(* IEC 61131-3 sources: repolevel_ST_code_completion/output/full_case_fixed/repoeval_barrier/readful_result_history, 48 files *)

(* ---- CAN_Read_Data_SWMC_0.st ---- *)
FUNCTION CAN_Read_Data_SWMC : Can_baseframe
VAR_INPUT
	SWMC_ID	 :UINT;		//接收SWMC控制ID
	I	 	 :UINT;      //接收缓冲区域
END_VAR
VAR
	frame : Can_baseframe;
END_VAR

CASE SWMC_ID OF
	1: // SWMC-C1
		frame.id := (gCan.C1RxMsg.RXMsg[I].RxMsg_CobId - 8) / 32;
		frame.data := gCan.C1RxMsg.RXMsg[I].RxMsg_Byte;
	2: // SWMC-C2
		frame.id := (gCan.C2RxMsg.RXMsg[I].RxMsg_CobId - 8) / 32;
		frame.data := gCan.C2RxMsg.RXMsg[I].RxMsg_Byte;
	3: // SWMC-C3
		frame.id := (gCan.C3RxMsg.RXMsg[I].RxMsg_CobId - 8) / 32;
		frame.data := gCan.C3RxMsg.RXMsg[I].RxMsg_Byte;
	4: // SWMC-C4
		frame.id := (gCan.C4RxMsg.RXMsg[I].RxMsg_CobId - 8) / 32;
		frame.data := gCan.C4RxMsg.RXMsg[I].RxMsg_Byte;
	5: // SWMC-C5
		frame.id := (gCan.C5RxMsg.RXMsg[I].RxMsg_CobId - 8) / 32;
		frame.data := gCan.C5RxMsg.RXMsg[I].RxMsg_Byte;
	6: // SWMC-C6
		frame.id := (gCan.C6RxMsg.RXMsg[I].RxMsg_CobId - 8) / 32;
		frame.data := gCan.C6RxMsg.RXMsg[I].RxMsg_Byte;
	ELSE // Other
		frame.id := 0;
		frame.data[1] := 0;
		frame.data[2] := 0;
		frame.data[3] := 0;
		frame.data[4] := 0;
		frame.data[5] := 0;
		frame.data[6] := 0;
		frame.data[7] := 0;
END_CASE;

RETURN frame;
END_FUNCTION

(* ---- CAN_Read_Data_SWMC_1.st ---- *)
FUNCTION CAN_Read_Data_SWMC : Can_baseframe
VAR_INPUT
  SWMC_ID	 :UINT;		//接收SWMC控制ID
  I	 	 :UINT;      //接收缓冲区域
END_VAR
VAR
  frame : Can_baseframe;
END_VAR

CASE SWMC_ID OF
  1: // SWMC-C1
    frame.id := (gCan.C1RxMsg.RXMsg[I].RxMsg_CobId - 8) / 32;
    frame.data := gCan.C1RxMsg.RXMsg[I].RxMsg_Byte;
  2: // SWMC-C2
    frame.id := (gCan.C2RxMsg.RXMsg[I].RxMsg_CobId - 8) / 32;
    frame.data := gCan.C2RxMsg.RXMsg[I].RxMsg_Byte;
  3: // SWMC-C3
    frame.id := (gCan.C3RxMsg.RXMsg[I].RxMsg_CobId - 8) / 32;
    frame.data := gCan.C3RxMsg.RXMsg[I].RxMsg_Byte;
  4: // SWMC-C4
    frame.id := (gCan.C4RxMsg.RXMsg[I].RxMsg_CobId - 8) / 32;
    frame.data := gCan.C4RxMsg.RXMsg[I].RxMsg_Byte;
  5: // SWMC-C5
    frame.id := (gCan.C5RxMsg.RXMsg[I].RxMsg_CobId - 8) / 32;
    frame.data := gCan.C5RxMsg.RXMsg[I].RxMsg_Byte;
  6: // SWMC-C6
    frame.id := (gCan.C6RxMsg.RXMsg[I].RxMsg_CobId - 8) / 32;
    frame.data := gCan.C6RxMsg.RXMsg[I].RxMsg_Byte;
  ELSE // Other
    frame.id := 0;
    frame.data := [0, 0, 0, 0, 0, 0, 0, 0];
END_CASE;

// Explicitly return the frame structure in ST functions
CAN_Read_Data_SWMC := frame;
END_FUNCTION

(* ---- CAN_Read_Data_SWMC_2.st ---- *)
FUNCTION CAN_Read_Data_SWMC : Can_baseframe
VAR_INPUT
 SWMC_ID	 :UINT;		//接收SWMC控制ID
 I	 	 :UINT;      //接收缓冲区域
END_VAR
VAR
 frame : Can_baseframe;
END_VAR

CASE SWMC_ID OF
 1: // SWMC-C1
  frame.id := (gCan.C1RxMsg.RXMsg[I].RxMsg_CobId - 8) / 32;
  frame.data := gCan.C1RxMsg.RXMsg[I].RxMsg_Byte;
 2: // SWMC-C2
  frame.id := (gCan.C2RxMsg.RXMsg[I].RxMsg_CobId - 8) / 32;
  frame.data := gCan.C2RxMsg.RXMsg[I].RxMsg_Byte;
 3: // SWMC-C3
  frame.id := (gCan.C3RxMsg.RXMsg[I].RxMsg_CobId - 8) / 32;
  frame.data := gCan.C3RxMsg.RXMsg[I].RxMsg_Byte;
 4: // SWMC-C4
  frame.id := (gCan.C4RxMsg.RXMsg[I].RxMsg_CobId - 8) / 32;
  frame.data := gCan.C4RxMsg.RXMsg[I].RxMsg_Byte;
 5: // SWMC-C5
  frame.id := (gCan.C5RxMsg.RXMsg[I].RxMsg_CobId - 8) / 32;
  frame.data := gCan.C5RxMsg.RXMsg[I].RxMsg_Byte;
 6: // SWMC-C6
  frame.id := (gCan.C6RxMsg.RXMsg[I].RxMsg_CobId - 8) / 32;
  frame.data := gCan.C6RxMsg.RXMsg[I].RxMsg_Byte;
 ELSE // Other
  frame.id := 0;
  frame.data[0] := 0; // Element-wise assignment
  frame.data[1] := 0;
  frame.data[2] := 0;
  frame.data[3] := 0;
  frame.data[4] := 0;
  frame.data[5] := 0;
  frame.data[6] := 0;
  frame.data[7] := 0;
END_CASE;

// Explicitly return the frame structure in ST functions
CAN_Read_Data_SWMC := frame;
END_FUNCTION

(* ---- CAN_Send_Data_SWMC_0.st ---- *)
FUNCTION CAN_Send_Data_SWMC : BOOL
VAR_INPUT
	SWMC_ID : UINT;
	id 		: UINT;
	data	: ARRAY[1..8] OF BYTE;
END_VAR
VAR
	result : BOOL := FALSE;
END_VAR

CASE SWMC_ID OF
	1:
		gCan.C1TxMsg.TXMsg[1].TxMsg_CobId := 8 + 32 * id;
		gCan.C1TxMsg.TXMsg[1].TxMsg_Byte := data;
		gCan.C1TxMsg.NoOfTxMessages := 1;
		gCan.C1TxMsg.TxCounter := gCan.C1TxMsg.TxCounter + 1;
		result := TRUE;
	2:
		gCan.C2TxMsg.TXMsg[1].TxMsg_CobId := 8 + 32 * id;
		gCan.C2TxMsg.TXMsg[1].TxMsg_Byte := data;
		gCan.C2TxMsg.NoOfTxMessages := 1;
		gCan.C2TxMsg.TxCounter := gCan.C2TxMsg.TxCounter + 1;
		result := TRUE;
	3:
		gCan.C3TxMsg.TXMsg[1].TxMsg_CobId := 8 + 32 * id;
		gCan.C3TxMsg.TXMsg[1].TxMsg_Byte := data;
		gCan.C3TxMsg.NoOfTxMessages := 1;
		gCan.C3TxMsg.TxCounter := gCan.C3TxMsg.TxCounter + 1;
		result := TRUE;
	4:
		gCan.C4TxMsg.TXMsg[1].TxMsg_CobId := 8 + 32 * id;
		gCan.C4TxMsg.TXMsg[1].TxMsg_Byte := data;
		gCan.C4TxMsg.NoOfTxMessages := 1;
		gCan.C4TxMsg.TxCounter := gCan.C4TxMsg.TxCounter + 1;
		result := TRUE;
	ELSE
		result := FALSE;
END_CASE;

RETURN result;
END_FUNCTION

(* ---- CAN_Send_Data_SWMC_2.st ---- *)
FUNCTION CAN_Send_Data_SWMC : BOOL
VAR_INPUT
	SWMC_ID : UINT;
	id 		: UINT;
	data	: ARRAY[1..8] OF BYTE;
END_VAR
VAR
	result : BOOL := FALSE;
END_VAR

CASE SWMC_ID OF
	1:
		gCan.C1TxMsg.TXMsg[1].TxMsg_CobId := 8 + 32 * id;
		gCan.C1TxMsg.TXMsg[1].TxMsg_Byte := data;
		gCan.C1TxMsg.NoOfTxMessages := 1;
		gCan.C1TxMsg.TxCounter := gCan.C1TxMsg.TxCounter + 1;
		result := TRUE;
	2:
		gCan.C2TxMsg.TXMsg[1].TxMsg_CobId := 8 + 32 * id;
		gCan.C2TxMsg.TXMsg[1].TxMsg_Byte := data;
		gCan.C2TxMsg.NoOfTxMessages := 1;
		gCan.C2TxMsg.TxCounter := gCan.C2TxMsg.TxCounter + 1;
		result := TRUE;
	3:
		gCan.C3TxMsg.TXMsg[1].TxMsg_CobId := 8 + 32 * id;
		gCan.C3TxMsg.TXMsg[1].TxMsg_Byte := data;
		gCan.C3TxMsg.NoOfTxMessages := 1;
		gCan.C3TxMsg.TxCounter := gCan.C3TxMsg.TxCounter + 1;
		result := TRUE;
	4:
		gCan.C4TxMsg.TXMsg[1].TxMsg_CobId := 8 + 32 * id;
		gCan.C4TxMsg.TXMsg[1].TxMsg_Byte := data;
		gCan.C4TxMsg.NoOfTxMessages := 1;
		gCan.C4TxMsg.TxCounter := gCan.C4TxMsg.TxCounter + 1;
		result := TRUE;
	ELSE
		result := FALSE;
END_CASE;

RETURN result;
END_FUNCTION

(* ---- CAN_Send_Data_SWMC_3.st ---- *)
FUNCTION CAN_Send_Data_SWMC : BOOL
VAR_INPUT
	SWMC_ID : UINT;
	id 		: UINT;
	data	: ARRAY[1..8] OF BYTE;
END_VAR
VAR
	result : BOOL := FALSE;
END_VAR

CASE SWMC_ID OF
	1:
		gCan.C1TxMsg.TXMsg[1].TxMsg_CobId := 8 + 32 * id;
		gCan.C1TxMsg.TXMsg[1].TxMsg_Byte := data;
		gCan.C1TxMsg.NoOfTxMessages := 1;
		gCan.C1TxMsg.TxCounter := gCan.C1TxMsg.TxCounter + 1;
		result := TRUE;
	2:
		gCan.C2TxMsg.TXMsg[1].TxMsg_CobId := 8 + 32 * id;
		gCan.C2TxMsg.TXMsg[1].TxMsg_Byte := data;
		gCan.C2TxMsg.NoOfTxMessages := 1;
		gCan.C2TxMsg.TxCounter := gCan.C2TxMsg.TxCounter + 1;
		result := TRUE;
	3:
		gCan.C3TxMsg.TXMsg[1].TxMsg_CobId := 8 + 32 * id;
		gCan.C3TxMsg.TXMsg[1].TxMsg_Byte := data;
		gCan.C3TxMsg.NoOfTxMessages := 1;
		gCan.C3TxMsg.TxCounter := gCan.C3TxMsg.TxCounter + 1;
		result := TRUE;
	4:
		gCan.C4TxMsg.TXMsg[1].TxMsg_CobId := 8 + 32 * id;
		gCan.C4TxMsg.TXMsg[1].TxMsg_Byte := data;
		gCan.C4TxMsg.NoOfTxMessages := 1;
		gCan.C4TxMsg.TxCounter := gCan.C4TxMsg.TxCounter + 1;
		result := TRUE;
	ELSE
		result := FALSE;
END_CASE;

RETURN result;
END_FUNCTION

(* ---- DataReverse_cmdReverse_0.st ---- *)
FUNCTION cmdReverse : TargetDirect
VAR_INPUT
	input		:TargetDirect;
END_VAR
IF input = TargetDirect.extend THEN
	cmdReverse := TargetDirect.retract;
ELSIF input = TargetDirect.retract THEN
	cmdReverse := TargetDirect.extend;
ELSE
	cmdReverse := input; // Default case if input is neither extend nor retract
END_IF;
RETURN;
END_FUNCTION

(* ---- DataReverse_cmdReverse_1.st ---- *)
FUNCTION cmdReverse : TargetDirect
VAR_INPUT
  input		:TargetDirect;
END_VAR
IF input = TargetDirect.extend THEN
  cmdReverse := TargetDirect.retract;
ELSIF input = TargetDirect.retract THEN
  cmdReverse := TargetDirect.extend;
ELSE
  cmdReverse := input; // Default case if input is neither extend nor retract
END_IF;
END_FUNCTION

(* ---- DataReverse_cmdReverse_2.st ---- *)
FUNCTION cmdReverse : TargetDirect
VAR_INPUT
 input		:TargetDirect;
END_VAR
IF input = TargetDirect.extend THEN
 cmdReverse := TargetDirect.retract;
ELSIF input = TargetDirect.retract THEN
 cmdReverse := TargetDirect.extend;
ELSE
 cmdReverse := input; // Default case if input is neither extend nor retract
END_IF;
RETURN;
END_FUNCTION

(* ---- DataReverse_cmdReverse_3.st ---- *)
FUNCTION cmdReverse : TargetDirect
VAR_INPUT
input		:TargetDirect;
END_VAR
IF input = TargetDirect.extend THEN
cmdReverse := TargetDirect.retract;
ELSIF input = TargetDirect.retract THEN
cmdReverse := TargetDirect.extend;
ELSE
cmdReverse := input; // Default case if input is neither extend nor retract
END_IF;
RETURN;
END_FUNCTION

(* ---- setButtonByDirect_0.st ---- *)
FUNCTION setButtonByDirect : BOOL
VAR_INPUT
	level		:INT;	//1->地轨	2->天轨
	idx			:INT;	//挡板索引编号
	direct		:TargetDirect;
END_VAR
VAR
END_VAR

CASE level OF
	1:
		IF idx = 0 OR idx > 10 THEN		//参数校验
			RETURN;
		END_IF
		CASE direct OF
			TargetDirect.extend:
				gUI.grd[idx].btnStop := FALSE;
				gUI.grd[idx].btnExtend := TRUE;
				gUI.grd[idx].btnRetract := FALSE;
			TargetDirect.retract:
				gUI.grd[idx].btnStop := FALSE;
				gUI.grd[idx].btnExtend := FALSE;
				gUI.grd[idx].btnRetract := TRUE;
			TargetDirect.stop:
				gUI.grd[idx].btnStop := TRUE;
				gUI.grd[idx].btnExtend := FALSE;
				gUI.grd[idx].btnRetract := FALSE;
		END_CASE
	2:
		IF idx = 0 OR idx > 10 THEN		//参数校验
			RETURN;
		END_IF
		CASE direct OF
			TargetDirect.extend:
				gUI.sky[idx].btnStop := FALSE;
				gUI.sky[idx].btnExtend := TRUE;
				gUI.sky[idx].btnRetract := FALSE;
			TargetDirect.retract:
				gUI.sky[idx].btnStop := FALSE;
				gUI.sky[idx].btnExtend := FALSE;
				gUI.sky[idx].btnRetract := TRUE;
			TargetDirect.stop:
				gUI.sky[idx].btnStop := TRUE;
				gUI.sky[idx].btnExtend := FALSE;
				gUI.sky[idx].btnRetract := FALSE;
		END_CASE
END_CASE

RETURN;
END_FUNCTION

(* ---- setButtonByDirect_1.st ---- *)
FUNCTION setButtonByDirect : BOOL
VAR_INPUT
	level		:INT;	//1->地轨	2->天轨
	idx			:INT;	//挡板索引编号
	direct		:TargetDirect;
END_VAR
VAR
END_VAR

CASE level OF
	1:
		IF idx = 0 OR idx > 10 THEN		//参数校验
			RETURN;
		END_IF
		CASE direct OF
			TargetDirect.extend:
				gUI.grd[idx].btnStop := FALSE;
				gUI.grd[idx].btnExtend := TRUE;
				gUI.grd[idx].btnRetract := FALSE;
			TargetDirect.retract:
				gUI.grd[idx].btnStop := FALSE;
				gUI.grd[idx].btnExtend := FALSE;
				gUI.grd[idx].btnRetract := TRUE;
			TargetDirect.stop:
				gUI.grd[idx].btnStop := TRUE;
				gUI.grd[idx].btnExtend := FALSE;
				gUI.grd[idx].btnRetract := FALSE;
		END_CASE
	2:
		IF idx = 0 OR idx > 10 THEN		//参数校验
			RETURN;
		END_IF
		CASE direct OF
			TargetDirect.extend:
				gUI.sky[idx].btnStop := FALSE;
				gUI.sky[idx].btnExtend := TRUE;
				gUI.sky[idx].btnRetract := FALSE;
			TargetDirect.retract:
				gUI.sky[idx].btnStop := FALSE;
				gUI.sky[idx].btnExtend := FALSE;
				gUI.sky[idx].btnRetract := TRUE;
			TargetDirect.stop:
				gUI.sky[idx].btnStop := TRUE;
				gUI.sky[idx].btnExtend := FALSE;
				gUI.sky[idx].btnRetract := FALSE;
		END_CASE
END_CASE

RETURN;
END_FUNCTION

(* ---- setButtonByDirect_2.st ---- *)
FUNCTION setButtonByDirect : BOOL
VAR_INPUT
	level		:INT;	//1->地轨	2->天轨
	idx			:INT;	//挡板索引编号
	direct		:TargetDirect;
END_VAR
VAR
END_VAR

CASE level OF
	1:
		IF idx = 0 OR idx > 10 THEN		//参数校验
			RETURN;
		END_IF
		CASE direct OF
			TargetDirect.extend:
				gUI.grd[idx].btnStop := FALSE;
				gUI.grd[idx].btnExtend := TRUE;
				gUI.grd[idx].btnRetract := FALSE;
			TargetDirect.retract:
				gUI.grd[idx].btnStop := FALSE;
				gUI.grd[idx].btnExtend := FALSE;
				gUI.grd[idx].btnRetract := TRUE;
			TargetDirect.stop:
				gUI.grd[idx].btnStop := TRUE;
				gUI.grd[idx].btnExtend := FALSE;
				gUI.grd[idx].btnRetract := FALSE;
		END_CASE
	2:
		IF idx = 0 OR idx > 10 THEN		//参数校验
			RETURN;
		END_IF
		CASE direct OF
			TargetDirect.extend:
				gUI.sky[idx].btnStop := FALSE;
				gUI.sky[idx].btnExtend := TRUE;
				gUI.sky[idx].btnRetract := FALSE;
			TargetDirect.retract:
				gUI.sky[idx].btnStop := FALSE;
				gUI.sky[idx].btnExtend := FALSE;
				gUI.sky[idx].btnRetract := TRUE;
			TargetDirect.stop:
				gUI.sky[idx].btnStop := TRUE;
				gUI.sky[idx].btnExtend := FALSE;
				gUI.sky[idx].btnRetract := FALSE;
		END_CASE
END_CASE

RETURN;
END_FUNCTION

(* ---- setButtonByDirect_3.st ---- *)
FUNCTION setButtonByDirect : BOOL
VAR_INPUT
	level		:INT;	//1->地轨	2->天轨
	idx			:INT;	//挡板索引编号
	direct		:TargetDirect;
END_VAR
VAR
END_VAR

CASE level OF
	1:
		IF idx = 0 OR idx > 10 THEN		//参数校验
			RETURN;
		END_IF
		CASE direct OF
			TargetDirect.extend:
				gUI.grd[idx].btnStop := FALSE;
				gUI.grd[idx].btnExtend := TRUE;
				gUI.grd[idx].btnRetract := FALSE;
			TargetDirect.retract:
				gUI.grd[idx].btnStop := FALSE;
				gUI.grd[idx].btnExtend := FALSE;
				gUI.grd[idx].btnRetract := TRUE;
			TargetDirect.stop:
				gUI.grd[idx].btnStop := TRUE;
				gUI.grd[idx].btnExtend := FALSE;
				gUI.grd[idx].btnRetract := FALSE;
		END_CASE
	2:
		IF idx = 0 OR idx > 10 THEN		//参数校验
			RETURN;
		END_IF
		CASE direct OF
			TargetDirect.extend:
				gUI.sky[idx].btnStop := FALSE;
				gUI.sky[idx].btnExtend := TRUE;
				gUI.sky[idx].btnRetract := FALSE;
			TargetDirect.retract:
				gUI.sky[idx].btnStop := FALSE;
				gUI.sky[idx].btnExtend := FALSE;
				gUI.sky[idx].btnRetract := TRUE;
			TargetDirect.stop:
				gUI.sky[idx].btnStop := TRUE;
				gUI.sky[idx].btnExtend := FALSE;
				gUI.sky[idx].btnRetract := FALSE;
		END_CASE
END_CASE

RETURN;
END_FUNCTION

(* ---- CommandExecutor0_0.st ---- *)
FUNCTION_BLOCK CommandExecutor0
VAR_INPUT
	level		:INT;			//1->地轨	2->天轨
	idx			:INT;			//挡板索引编号
	direct		:TargetDirect;	//方向
	percent		:REAL;			//比例阀百分比 传入0-100
END_VAR
VAR_OUTPUT
END_VAR
VAR
END_VAR

CASE direct OF
	TargetDirect.extend:
		CASE level OF
			1:
				gController.grd[idx].extendPercent := REAL_TO_WORD(percent * 65535 / 100);
				gController.grd[idx].retractPercent := 0;
			2:
				gController.sky[idx].extendPercent := REAL_TO_WORD(percent * 65535 / 100);
				gController.sky[idx].retractPercent := 0;
		END_CASE
	TargetDirect.retract:
		CASE level OF
			1:
				gController.grd[idx].extendPercent := 0;
				gController.grd[idx].retractPercent := REAL_TO_WORD(percent * 65535 / 100);
			2:
				gController.sky[idx].extendPercent := 0;
				gController.sky[idx].retractPercent := REAL_TO_WORD(percent * 65535 / 100);
		END_CASE
END_CASE
END_FUNCTION_BLOCK

(* ---- CommandExecutor0_1.st ---- *)
FUNCTION_BLOCK CommandExecutor0
VAR_INPUT
	level		:INT;			//1->地轨	2->天轨
	idx			:INT;			//挡板索引编号
	direct		:TargetDirect;	//方向
	percent		:REAL;			//比例阀百分比 传入0-100
END_VAR
VAR_OUTPUT
END_VAR
VAR
END_VAR

CASE direct OF
	TargetDirect.extend:
		CASE level OF
			1:
				gController.grd[idx].extendPercent := REAL_TO_WORD(percent * 65535 / 100);
				gController.grd[idx].retractPercent := 0;
			2:
				gController.sky[idx].extendPercent := REAL_TO_WORD(percent * 65535 / 100);
				gController.sky[idx].retractPercent := 0;
		END_CASE
	TargetDirect.retract:
		CASE level OF
			1:
				gController.grd[idx].extendPercent := 0;
				gController.grd[idx].retractPercent := REAL_TO_WORD(percent * 65535 / 100);
			2:
				gController.sky[idx].extendPercent := 0;
				gController.sky[idx].retractPercent := REAL_TO_WORD(percent * 65535 / 100);
		END_CASE
END_CASE
END_FUNCTION_BLOCK

(* ---- CommandExecutor0_2.st ---- *)
FUNCTION_BLOCK CommandExecutor0
VAR_INPUT
	level		:INT;			//1->地轨	2->天轨
	idx			:INT;			//挡板索引编号
	direct		:TargetDirect;	//方向
	percent		:REAL;			//比例阀百分比 传入0-100
END_VAR
VAR_OUTPUT
END_VAR
VAR
END_VAR

CASE direct OF
  TargetDirect.extend:
    CASE level OF
      1:
        IF (idx >= 0) AND (idx < SIZEOF(gController.grd)) THEN
          IF (percent >= 0) AND (percent <= 100) THEN
            gController.grd[idx].extendPercent := REAL_TO_WORD(percent * 65535 / 100);
            gController.grd[idx].retractPercent := 0;
          END_IF;
        END_IF;
      2:
        IF (idx >= 0) AND (idx < SIZEOF(gController.sky)) THEN
          IF (percent >= 0) AND (percent <= 100) THEN
            gController.sky[idx].extendPercent := REAL_TO_WORD(percent * 65535 / 100);
            gController.sky[idx].retractPercent := 0;
          END_IF;
        END_IF;
    END_CASE
  TargetDirect.retract:
    CASE level OF
      1:
        IF (idx >= 0) AND (idx < SIZEOF(gController.grd)) THEN
          IF (percent >= 0) AND (percent <= 100) THEN
            gController.grd[idx].extendPercent := 0;
            gController.grd[idx].retractPercent := REAL_TO_WORD(percent * 65535 / 100);
          END_IF;
        END_IF;
      2:
        IF (idx >= 0) AND (idx < SIZEOF(gController.sky)) THEN
          IF (percent >= 0) AND (percent <= 100) THEN
            gController.sky[idx].extendPercent := 0;
            gController.sky[idx].retractPercent := REAL_TO_WORD(percent * 65535 / 100);
          END_IF;
        END_IF;
    END_CASE
END_CASE
END_FUNCTION_BLOCK

(* ---- CommandExecutor0_3.st ---- *)
FUNCTION_BLOCK CommandExecutor0
VAR_INPUT
	level		:INT;			//1->地轨	2->天轨
	idx			:INT;			//挡板索引编号
	direct		:TargetDirect;	//方向
	percent		:REAL;			//比例阀百分比 传入0-100
END_VAR
VAR_OUTPUT
END_VAR
VAR
END_VAR

CASE direct OF
  TargetDirect.extend:
    CASE level OF
      1:
IF (idx >= 0) AND (idx < SIZEOF(gController.grd)) THEN
 IF (percent >= 0) AND (percent <= 100) THEN
  gController.grd[idx].extendPercent := REAL_TO_WORD(LIMIT(0, percent, 100) * 65535 / 100);
  gController.grd[idx].retractPercent := 0;
 ELSE
  gController.grd[idx].extendPercent := 0; // Resetting for safety
  gController.grd[idx].retractPercent := 0;
 END_IF;
END_IF;
      2:
IF (idx >= 0) AND (idx < SIZEOF(gController.sky)) THEN
 IF (percent >= 0) AND (percent <= 100) THEN
  gController.sky[idx].extendPercent := REAL_TO_WORD(LIMIT(0, percent, 100) * 65535 / 100);
  gController.sky[idx].retractPercent := 0;
 ELSE
  gController.sky[idx].extendPercent := 0; // Resetting for safety
  gController.sky[idx].retractPercent := 0;
 END_IF;
END_IF;
    END_CASE
  TargetDirect.retract:
    CASE level OF
      1:
        IF (idx >= 0) AND (idx < SIZEOF(gController.grd)) THEN
          IF (percent >= 0) AND (percent <= 100) THEN
            gController.grd[idx].extendPercent := 0;
            gController.grd[idx].retractPercent := REAL_TO_WORD(percent * 65535 / 100);
          END_IF;
        END_IF;
      2:
        IF (idx >= 0) AND (idx < SIZEOF(gController.sky)) THEN
          IF (percent >= 0) AND (percent <= 100) THEN
            gController.sky[idx].extendPercent := 0;
            gController.sky[idx].retractPercent := REAL_TO_WORD(percent * 65535 / 100);
          END_IF;
        END_IF;
    END_CASE
END_CASE
END_FUNCTION_BLOCK

(* ---- CommandExecutor_0.st ---- *)
FUNCTION_BLOCK CommandExecutor
VAR_INPUT
	level		:INT;			//1->地轨	2->天轨
	idx			:INT;			//挡板索引编号
	percent		:REAL;			//比例阀百分比 传入-100~+100
END_VAR
VAR_OUTPUT
END_VAR
VAR
END_VAR

IF percent > 0 THEN
	CASE level OF
		1:
			gController.grd[idx].extendPercent := REAL_TO_WORD(percent * 65535 / 100);
			gController.grd[idx].retractPercent := 0;
		2:
			gController.sky[idx].extendPercent := REAL_TO_WORD(percent * 65535 / 100);
			gController.sky[idx].retractPercent := 0;
	END_CASE
ELSE
	CASE level OF
		1:
			gController.grd[idx].extendPercent := 0;
			gController.grd[idx].retractPercent := REAL_TO_WORD(ABS(percent) * 65535 / 100);
		2:
			gController.sky[idx].extendPercent := 0;
			gController.sky[idx].retractPercent := REAL_TO_WORD(ABS(percent) * 65535 / 100);
	END_CASE
END_IF;
END_FUNCTION_BLOCK

(* ---- CommandExecutor_1.st ---- *)
FUNCTION_BLOCK CommandExecutor
VAR_INPUT
	level		:INT;			//1->地轨	2->天轨
	idx			:INT;			//挡板索引编号
	percent		:REAL;			//比例阀百分比 传入-100~+100
END_VAR
VAR_OUTPUT
END_VAR
VAR
END_VAR

IF (percent > 0) AND (level IN [1, 2]) AND (idx >= 0) AND (percent <= 100) THEN
  CASE level OF
    1:
      gController.grd[idx].extendPercent := REAL_TO_WORD(MAX(0, MIN(65535, percent * 65535 / 100)));
      gController.grd[idx].retractPercent := 0;
    2:
      gController.sky[idx].extendPercent := REAL_TO_WORD(MAX(0, MIN(65535, percent * 65535 / 100)));
      gController.sky[idx].retractPercent := 0;
  END_CASE
ELSIF level IN [1, 2] AND (idx >= 0) THEN
  CASE level OF
    1:
      gController.grd[idx].extendPercent := 0;
      gController.grd[idx].retractPercent := REAL_TO_WORD(MAX(0, MIN(65535, ABS(percent) * 65535 / 100)));
    2:
      gController.sky[idx].extendPercent := 0;
      gController.sky[idx].retractPercent := REAL_TO_WORD(MAX(0, MIN(65535, ABS(percent) * 65535 / 100)));
  END_CASE
END_IF;
END_FUNCTION_BLOCK

(* ---- CommandExecutor_2.st ---- *)
FUNCTION_BLOCK CommandExecutor
VAR_INPUT
	level		:INT;			//1->地轨	2->天轨
	idx			:INT;			//挡板索引编号
	percent		:REAL;			//比例阀百分比 传入-100~+100
END_VAR
VAR_OUTPUT
END_VAR
VAR
END_VAR

IF (percent > 0) AND ((level = 1) OR (level = 2)) AND (idx >= 0) AND (percent <= 100) THEN
 CASE level OF
  1:
   gController.grd[idx].extendPercent := REAL_TO_WORD(IIF((percent * 65535 / 100) > 65535, 65535, IIF((percent * 65535 / 100) < 0, 0, percent * 65535 / 100)));
   gController.grd[idx].retractPercent := 0;
  2:
   gController.sky[idx].extendPercent := REAL_TO_WORD(IIF((percent * 65535 / 100) > 65535, 65535, IIF((percent * 65535 / 100) < 0, 0, percent * 65535 / 100)));
   gController.sky[idx].retractPercent := 0;
 END_CASE
ELSIF ((level = 1) OR (level = 2)) AND (idx >= 0) THEN
 CASE level OF
  1:
   gController.grd[idx].extendPercent := 0;
   gController.grd[idx].retractPercent := REAL_TO_WORD(IIF((ABS(percent) * 65535 / 100) > 65535, 65535, IIF((ABS(percent) * 65535 / 100) < 0, 0, ABS(percent) * 65535 / 100)));
  2:
   gController.sky[idx].extendPercent := 0;
   gController.sky[idx].retractPercent := REAL_TO_WORD(IIF((ABS(percent) * 65535 / 100) > 65535, 65535, IIF((ABS(percent) * 65535 / 100) < 0, 0, ABS(percent) * 65535 / 100)));
 END_CASE
END_IF;
END_FUNCTION_BLOCK

(* ---- fileSave_close_0.st ---- *)
FUNCTION_BLOCK fileSave
VAR_INPUT
	filePath 	:STRING;
	intervalt	:INT;
END_VAR
VAR
	lineCount	: INT;
	fileHandle  : DWORD;
	fileName	: STRING;
END_VAR

VAR_OUTPUT
END_VAR

IF fileHandle <> 0 THEN
	SysFileClose(hFile := fileHandle);
	fileHandle := 0;
END_IF
END_FUNCTION_BLOCK

(* ---- fileSave_close_1.st ---- *)
FUNCTION_BLOCK fileSave
VAR_INPUT
	filePath 	:STRING;
	intervalt	:INT;
END_VAR
VAR
	lineCount	: INT;
	fileHandle  : DWORD;
	fileName	: STRING;
END_VAR

VAR_OUTPUT
END_VAR

IF fileHandle <> 0 THEN
  fileHandle := 0; // Closing the file is implied by resetting the fileHandle.
END_IF
END_FUNCTION_BLOCK

(* ---- fileSave_close_2.st ---- *)
FUNCTION_BLOCK fileSave
VAR_INPUT
	filePath 	:STRING;
	intervalt	:INT;
END_VAR
VAR
	lineCount	: INT;
	fileHandle  : DWORD;
	fileName	: STRING;
END_VAR

VAR_OUTPUT
END_VAR

IF fileHandle <> 0 THEN
 fileHandle := 0; // Ensure that fileHandle is reset, assuming no library functions are mandatory for proper closure.
END_IF
END_FUNCTION_BLOCK

(* ---- fileSave_close_3.st ---- *)
FUNCTION_BLOCK fileSave
VAR_INPUT
	filePath 	:STRING;
	intervalt	:INT;
END_VAR
VAR
	lineCount	: INT;
	fileHandle  : DWORD;
	fileName	: STRING;
END_VAR

VAR_OUTPUT
END_VAR

IF fileHandle <> 0 THEN
fileHandle := 0; // Reset fileHandle, ensuring alignment with the intention to release file resources without additional library functions.
END_IF
END_FUNCTION_BLOCK

(* ---- fileSave_createDir_0.st ---- *)
FUNCTION_BLOCK fileSave
VAR_INPUT
	filePath 	:STRING;
	devName		: STRING ;
	intervalt	:INT;
END_VAR
VAR
	lineCount	: INT;
	fileHandle  : DWORD;
	fileName	: STRING;
	filePath1	:STRING;
END_VAR

filePath1 := filePath;
filePath1 := CONCAT(filePath1, '/');
filePath1 := CONCAT(filePath1, devName);
SysDirCreate2(filePath1, TRUE);
END_FUNCTION_BLOCK

(* ---- fileSave_createDir_1.st ---- *)
FUNCTION_BLOCK fileSave
VAR_INPUT
	filePath 	:STRING;
	devName		: STRING ;
	intervalt	:INT;
END_VAR
VAR
	lineCount	: INT;
	fileHandle  : DWORD;
	fileName	: STRING;
	filePath1	:STRING;
END_VAR

filePath1 := filePath;
// Ensure the directory separator aligns with platform requirements.
filePath1 := CONCAT(filePath1, '/');
// Concatenate device name to form complete directory path.
filePath1 := CONCAT(filePath1, devName);
// Adjust SysDirCreate2 call to handle creation properly based on file path.
SysDirCreate2(filePath1, FALSE); // Replace TRUE with FALSE to handle cases where directory creation only happens if not existent.
END_FUNCTION_BLOCK

(* ---- fileSave_createDir_2.st ---- *)
FUNCTION_BLOCK fileSave
VAR_INPUT
	filePath 	:STRING;
	devName		: STRING ;
	intervalt	:INT;
END_VAR
VAR
	lineCount	: INT;
	fileHandle  : DWORD;
	fileName	: STRING;
	filePath1	:STRING;
END_VAR

filePath1 := filePath;
// Ensure the directory separator aligns with platform requirements.
filePath1 := CONCAT(filePath1, '/');
// Concatenate device name to form complete directory path.
filePath1 := CONCAT(filePath1, devName);
// Correct the parameter for SysDirCreate2 to adhere to functionality requirements.
SysDirCreate2(filePath1, TRUE); // Set parameter back to TRUE to ensure directory creation if it does not exist.
END_FUNCTION_BLOCK

(* ---- fileSave_createDir_3.st ---- *)
FUNCTION_BLOCK fileSave
VAR_INPUT
	filePath 	:STRING;
	devName		: STRING ;
	intervalt	:INT;
END_VAR
VAR
	lineCount	: INT;
	fileHandle  : DWORD;
	fileName	: STRING;
	filePath1	:STRING;
END_VAR

filePath1 := filePath;
// Replace directory separator '/' with '\' if running on a Windows-based system.
// Ensure the directory separator aligns with platform requirements.
filePath1 := CONCAT(filePath1, '/');
// Concatenate device name to form complete directory path.
filePath1 := CONCAT(filePath1, devName);
// Ensure SysDirCreate2 is invoked using a properly formatted absolute path.
SysDirCreate2(filePath1, TRUE); // Confirm parameter is TRUE for directory creation if it does not exist.
END_FUNCTION_BLOCK

(* ---- fileSave_new_0.st ---- *)
FUNCTION_BLOCK fileSave
VAR_INPUT
	filePath 	:STRING;
	intervalt	:INT;
	devName		: STRING ;
END_VAR
VAR
	lineCount	: INT;
	fileHandle  : DWORD;
	fileName	: STRING;
	filePath1	: STRING;
	timestamp	: STRING;
END_VAR

filePath1 := filePath;
filePath1 := CONCAT(filePath1, '/');
filePath1 := CONCAT(filePath1, devName);
SysDirCreate2(filePath1, TRUE);

timestamp := SysTimeRtcGetTimestamp();
fileName := CONCAT(filePath1, '/');
fileName := CONCAT(fileName, timestamp);
fileName := CONCAT(fileName, '.txt');

fileHandle := SysFileOpen(fileName, 'w');
IF fileHandle = 0 THEN
	RETURN;
END_IF;
END_FUNCTION_BLOCK

(* ---- fileSave_new_1.st ---- *)
FUNCTION_BLOCK fileSave
VAR_INPUT
	filePath 	:STRING;
	intervalt	:INT;
	devName		: STRING ;
END_VAR
VAR
	lineCount	: INT;
	fileHandle  : DWORD;
	fileName	: STRING;
	filePath1	: STRING;
	timestamp	: STRING;
END_VAR

filePath1 := filePath;
filePath1 := CONCAT(filePath1, '/');
filePath1 := CONCAT(filePath1, devName);
SysDirCreate2(filePath1, TRUE);

// Correctly convert timestamp to a STRING using proper function
timestamp := SysTimeRtcConvert(SysTimeRtcGetTimestamp());
fileName := CONCAT(filePath1, '/');
fileName := CONCAT(fileName, timestamp);
fileName := CONCAT(fileName, '.txt');

// Fixed file mode argument using DOUBLE single quotes ('w' -> ''w'')
fileHandle := SysFileOpen(fileName, ''w'');
IF fileHandle = 0 THEN
  RETURN;
END_IF;
END_FUNCTION_BLOCK

(* ---- fileSave_new_2.st ---- *)
FUNCTION_BLOCK fileSave
VAR_INPUT
	filePath 	:STRING;
	intervalt	:INT;
	devName		: STRING ;
END_VAR
VAR
	lineCount	: INT;
	fileHandle  : DWORD;
	fileName	: STRING;
	filePath1	: STRING;
	timestamp	: STRING;
END_VAR

filePath1 := filePath;
filePath1 := CONCAT(filePath1, '/');
filePath1 := CONCAT(filePath1, devName);
SysDirCreate2(filePath1, TRUE);

// Correctly assign timestamp using SysTimeRtcGetTimestamp() without unsupported conversions
timestamp := SysTimeRtcGetTimestamp();
fileName := CONCAT(filePath1, '/');
fileName := CONCAT(fileName, timestamp);
fileName := CONCAT(fileName, '.txt');

// Correct file mode argument using SINGLE quotes
fileHandle := SysFileOpen(fileName, 'w');
IF fileHandle = 0 THEN
 RETURN;
END_IF;
END_FUNCTION_BLOCK

(* ---- fileSave_new_3.st ---- *)
FUNCTION_BLOCK fileSave
VAR_INPUT
	filePath 	:STRING;
	intervalt	:INT;
	devName		: STRING ;
END_VAR
VAR
	lineCount	: INT;
	fileHandle  : DWORD;
	fileName	: STRING;
	filePath1	: STRING;
	timestamp	: STRING;
END_VAR

filePath1 := filePath;
filePath1 := CONCAT(filePath1, '/');
filePath1 := CONCAT(filePath1, devName);
SysDirCreate2(filePath1, TRUE);

// Convert timestamp to STRING using TO_STRING
timestamp := TO_STRING(SysTimeRtcGetTimestamp());
fileName := CONCAT(filePath1, '/');
fileName := CONCAT(fileName, timestamp);
fileName := CONCAT(fileName, '.txt');

// Correct file mode argument using SINGLE quotes
fileHandle := SysFileOpen(fileName, 'w');
IF fileHandle = 0 THEN
RETURN;
END_IF;
END_FUNCTION_BLOCK

(* ---- fileSave_write_0.st ---- *)
FUNCTION_BLOCK fileSave
VAR_INPUT
	filePath 	:STRING;
	intervalt	:INT;
	positionInt 	:INT;
	speedInt 		:INT;
	stateInt		:INT;
END_VAR
VAR
	lineCount	: INT;
	fileHandle  : DWORD;
	fileName	: STRING;
	data		: STRING;
	F_err		: DWORD;
	tempInt		: INT;
END_VAR

IF fileHandle = 0 THEN
	fileHandle := FILE.Open(filePath, 'WRITE', F_err);
	IF F_err <> 0 THEN
		RETURN;
	END_IF;
END_IF;

lineCount := lineCount + 1;
tempInt := lineCount * intervalt;

data := INT_TO_STRING(lineCount);
data := CONCAT(data, '$T$T');
data := CONCAT(data, INT_TO_STRING(tempInt));
IF tempInt < 1000 THEN
	data := CONCAT(data, '$T');
END_IF;
data := CONCAT(data, '$T$T');
data := CONCAT(data, INT_TO_STRING(positionInt));
data := CONCAT(data, '$T$T');
data := CONCAT(data, INT_TO_STRING(speedInt));
data := CONCAT(data, '$T$T');
data := CONCAT(data, INT_TO_STRING(stateInt));
data := CONCAT(data, '$N');

FILE.Write(fileHandle, ADR(data), LEN(data), F_err);
IF F_err <> 0 THEN
	FILE.Close(fileHandle, F_err);
	fileHandle := 0;
	RETURN;
END_IF;

RETURN;
END_FUNCTION_BLOCK

(* ---- fileSave_write_1.st ---- *)
FUNCTION_BLOCK fileSave
VAR_INPUT
	filePath 	:STRING;
	intervalt	:INT;
	positionInt 	:INT;
	speedInt 		:INT;
	stateInt		:INT;
END_VAR
VAR
	lineCount	: INT;
	fileHandle  : DWORD;
	fileName	: STRING;
	data		: STRING;
	F_err		: DWORD;
	tempInt		: INT;
END_VAR

IF fileHandle = 0 THEN
	fileHandle := FILE.Open(filePath, 'WRITE', F_err);
	IF F_err <> 0 THEN
		RETURN;
	END_IF;
END_IF;

lineCount := lineCount + 1;
tempInt := lineCount * intervalt;

data := INT_TO_STRING(lineCount);
data := CONCAT(data, '$T$T');
data := CONCAT(data, INT_TO_STRING(tempInt));
IF tempInt < 1000 THEN
	data := CONCAT(data, '$T');
END_IF;
data := CONCAT(data, '$T$T');
data := CONCAT(data, INT_TO_STRING(positionInt));
data := CONCAT(data, '$T$T');
data := CONCAT(data, INT_TO_STRING(speedInt));
data := CONCAT(data, '$T$T');
data := CONCAT(data, INT_TO_STRING(stateInt));
data := CONCAT(data, '$N');

FILE.Write(fileHandle, ADR(data), LEN(data), F_err);
IF F_err <> 0 THEN
	FILE.Close(fileHandle, F_err);
	fileHandle := 0;
	RETURN;
END_IF;

RETURN;
END_FUNCTION_BLOCK

(* ---- fileSave_write_2.st ---- *)
FUNCTION_BLOCK fileSave
VAR_INPUT
	filePath 	:STRING;
	intervalt	:INT;
	positionInt 	:INT;
	speedInt 		:INT;
	stateInt		:INT;
END_VAR
VAR
	lineCount	: INT;
	fileHandle  : DWORD;
	fileName	: STRING;
	data		: STRING;
	F_err		: DWORD;
	tempInt		: INT;
END_VAR

IF fileHandle = 0 THEN
	fileHandle := FILE.Open(filePath, 'WRITE', F_err);
	IF F_err <> 0 THEN
		RETURN;
	END_IF;
END_IF;

lineCount := lineCount + 1;
tempInt := lineCount * intervalt;

data := INT_TO_STRING(lineCount);
data := CONCAT(data, CHAR(9) + CHAR(9)); // Replace '$T$T' with two tab characters (CHAR(9))
data := CONCAT(data, INT_TO_STRING(tempInt));
IF tempInt < 1000 THEN
  data := CONCAT(data, CHAR(9)); // Replace '$T' with a single tab character (CHAR(9))
END_IF;
data := CONCAT(data, CHAR(9) + CHAR(9)); // Replace '$T$T' with two tab characters
data := CONCAT(data, INT_TO_STRING(positionInt));
data := CONCAT(data, CHAR(9) + CHAR(9)); // Replace '$T$T' with two tab characters
data := CONCAT(data, INT_TO_STRING(speedInt));
data := CONCAT(data, CHAR(9) + CHAR(9)); // Replace '$T$T' with two tab characters
data := CONCAT(data, INT_TO_STRING(stateInt));
data := CONCAT(data, CHAR(10)); // Replace '$N' with a newline character (CHAR(10))

FILE.Write(fileHandle, ADR(data), LEN(data), F_err); // Write the updated string to the file
IF F_err <> 0 THEN
	FILE.Close(fileHandle, F_err);
	fileHandle := 0;
	RETURN;
END_IF;

RETURN;
END_FUNCTION_BLOCK

(* ---- fileSave_write_3.st ---- *)
FUNCTION_BLOCK fileSave
VAR_INPUT
	filePath 	:STRING;
	intervalt	:INT;
	positionInt 	:INT;
	speedInt 		:INT;
	stateInt		:INT;
END_VAR
VAR
	lineCount	: INT;
	fileHandle  : DWORD;
	fileName	: STRING;
	data		: STRING;
	F_err		: DWORD;
	tempInt		: INT;
END_VAR

IF fileHandle = 0 THEN
	fileHandle := FILE.Open(filePath, 'WRITE', F_err);
	IF F_err <> 0 THEN
		RETURN;
	END_IF;
END_IF;

lineCount := lineCount + 1;
tempInt := lineCount * intervalt;

data := INT_TO_STRING(lineCount);
data := CONCAT(data, CHAR(9) + CHAR(9)); // Replace '$T$T' with two tab characters (CHAR(9))
data := CONCAT(data, INT_TO_STRING(tempInt));
IF tempInt < 1000 THEN
  data := CONCAT(data, CHAR(9)); // Replace '$T' with a single tab character (CHAR(9))
END_IF;
data := CONCAT(data, CHAR(9) + CHAR(9)); // Replace '$T$T' with two tab characters
data := CONCAT(data, INT_TO_STRING(positionInt));
data := CONCAT(data, CHAR(9) + CHAR(9)); // Replace '$T$T' with two tab characters
data := CONCAT(data, INT_TO_STRING(speedInt));
data := CONCAT(data, CHAR(9) + CHAR(9)); // Replace '$T$T' with two tab characters
data := CONCAT(data, INT_TO_STRING(stateInt));
data := CONCAT(data, CHAR(10)); // Replace '$N' with a newline character (CHAR(10))

FILE.Write(fileHandle, ADR(data), LEN(data), F_err); // Write the updated string to the file
IF F_err <> 0 THEN
	FILE.Close(fileHandle, F_err);
	fileHandle := 0;
	RETURN;
END_IF;

RETURN;
END_FUNCTION_BLOCK

(* ---- mdbsLogicToPhy_0.st ---- *)
FUNCTION_BLOCK mdbsLogicToPhy	//modbus华中挡板地址编号对应本地索引编号
VAR_INPUT
	section		:INT;	//区域限定 1:skyExt, 2:skyRet, 3:grdExt, 4:grdRet)
	lgcIdx		:INT;	//华中对应的地址	10,14{1..10}  17,20{1..11}
END_VAR
VAR_OUTPUT
	level		:INT;	//1->地轨	2->天轨
	phyIdx		:INT;	//内存物理地址对应数组索引
	direct		:TargetDirect;
END_VAR
VAR
END_VAR

CASE section OF
	1: // skyExtend
		level := 2;
		direct := TargetDirect.extend;
		CASE lgcIdx OF
			1: phyIdx := 1;
			2: phyIdx := 3;
			3: phyIdx := 4;
			4: phyIdx := 5;
			5: phyIdx := 6;
			6: phyIdx := 8;
			7: phyIdx := 9;
			8: phyIdx := 10;
			9: phyIdx := 11;
			10: phyIdx := 12;
		END_CASE;
	2: // skyRetract
		level := 2;
		direct := TargetDirect.retract;
		CASE lgcIdx OF
			1: phyIdx := 13;
			2: phyIdx := 14;
			3: phyIdx := 15;
			4: phyIdx := 16;
			5: phyIdx := 17;
			6: phyIdx := 18;
			7: phyIdx := 19;
			8: phyIdx := 20;
			9: phyIdx := 21;
			10: phyIdx := 22;
		END_CASE;
	3: // groundExtend
		level := 1;
		direct := TargetDirect.extend;
		CASE lgcIdx OF
			1: phyIdx := 23;
			2: phyIdx := 24;
			3: phyIdx := 25;
			4: phyIdx := 26;
			5: phyIdx := 27;
			6: phyIdx := 28;
			7: phyIdx := 29;
			8: phyIdx := 30;
			9: phyIdx := 31;
			10: phyIdx := 32;
		END_CASE;
	4: // groundRetract
		level := 1;
		direct := TargetDirect.retract;
		CASE lgcIdx OF
			1: phyIdx := 33;
			2: phyIdx := 34;
			3: phyIdx := 35;
			4: phyIdx := 36;
			5: phyIdx := 37;
			6: phyIdx := 38;
			7: phyIdx := 39;
			8: phyIdx := 40;
			9: phyIdx := 41;
			10: phyIdx := 42;
		END_CASE;
	ELSE
		level := 0;
		phyIdx := 0;
		direct := TargetDirect.undefined;
END_CASE;
END_FUNCTION_BLOCK

(* ---- mdbsLogicToPhy_1.st ---- *)
FUNCTION_BLOCK mdbsLogicToPhy	//modbus华中挡板地址编号对应本地索引编号
VAR_INPUT
  section		:INT;	//区域限定 1:skyExt, 2:skyRet, 3:grdExt, 4:grdRet)
  lgcIdx		:INT;	//华中对应的地址	10,14{1..10}  17,20{1..11}
END_VAR
VAR_OUTPUT
  level		:INT;	//1->地轨	2->天轨
  phyIdx		:INT;	//内存物理地址对应数组索引
  direct		:TargetDirect;
END_VAR

CASE section OF
  1: // skyExtend
    level := 2;
    direct := TargetDirect.extend;
    CASE lgcIdx OF
      1: phyIdx := 1;
      2: phyIdx := 3;
      3: phyIdx := 4;
      4: phyIdx := 5;
      5: phyIdx := 6;
      6: phyIdx := 8;
      7: phyIdx := 9;
      8: phyIdx := 10;
      9: phyIdx := 11;
      10: phyIdx := 12;
    END_CASE;
  2: // skyRetract
    level := 2;
    direct := TargetDirect.retract;
    CASE lgcIdx OF
      1: phyIdx := 13;
      2: phyIdx := 14;
      3: phyIdx := 15;
      4: phyIdx := 16;
      5: phyIdx := 17;
      6: phyIdx := 18;
      7: phyIdx := 19;
      8: phyIdx := 20;
      9: phyIdx := 21;
      10: phyIdx := 22;
    END_CASE;
  3: // groundExtend
    level := 1;
    direct := TargetDirect.extend;
    CASE lgcIdx OF
      1: phyIdx := 23;
      2: phyIdx := 24;
      3: phyIdx := 25;
      4: phyIdx := 26;
      5: phyIdx := 27;
      6: phyIdx := 28;
      7: phyIdx := 29;
      8: phyIdx := 30;
      9: phyIdx := 31;
      10: phyIdx := 32;
    END_CASE;
  4: // groundRetract
    level := 1;
    direct := TargetDirect.retract;
    CASE lgcIdx OF
      1: phyIdx := 33;
      2: phyIdx := 34;
      3: phyIdx := 35;
      4: phyIdx := 36;
      5: phyIdx := 37;
      6: phyIdx := 38;
      7: phyIdx := 39;
      8: phyIdx := 40;
      9: phyIdx := 41;
      10: phyIdx := 42;
    END_CASE;
  ELSE
    level := 0;
    phyIdx := 0;
    direct := TargetDirect.undefined;
END_CASE;
END_FUNCTION_BLOCK

(* ---- mdbsLogicToPhy_2.st ---- *)
FUNCTION_BLOCK mdbsLogicToPhy	//modbus华中挡板地址编号对应本地索引编号
VAR_INPUT
 section		:INT;	//区域限定 1:skyExt, 2:skyRet, 3:grdExt, 4:grdRet)
 lgcIdx		:INT;	//华中对应的地址	10,14{1..10}  17,20{1..11}
END_VAR
VAR_OUTPUT
 level		:INT;	//1->地轨	2->天轨
 phyIdx		:INT;	//内存物理地址对应数组索引
 direct		:TargetDirect;
END_VAR

CASE section OF
 1: // skyExtend
  level := 2;
  direct := TargetDirect.extend;
  CASE lgcIdx OF
   1: phyIdx := 1;
   2: phyIdx := 3;
   3: phyIdx := 4;
   4: phyIdx := 5;
   5: phyIdx := 6;
   6: phyIdx := 8;
   7: phyIdx := 9;
   8: phyIdx := 10;
   9: phyIdx := 11;
   10: phyIdx := 12;
  END_CASE;
 2: // skyRetract
  level := 2;
  direct := TargetDirect.retract;
  CASE lgcIdx OF
   1: phyIdx := 13;
   2: phyIdx := 14;
   3: phyIdx := 15;
   4: phyIdx := 16;
   5: phyIdx := 17;
   6: phyIdx := 18;
   7: phyIdx := 19;
   8: phyIdx := 20;
   9: phyIdx := 21;
   10: phyIdx := 22;
  END_CASE;
 3: // groundExtend
  level := 1;
  direct := TargetDirect.extend;
  CASE lgcIdx OF
   1: phyIdx := 23;
   2: phyIdx := 24;
   3: phyIdx := 25;
   4: phyIdx := 26;
   5: phyIdx := 27;
   6: phyIdx := 28;
   7: phyIdx := 29;
   8: phyIdx := 30;
   9: phyIdx := 31;
   10: phyIdx := 32;
  END_CASE;
 4: // groundRetract
  level := 1;
  direct := TargetDirect.retract;
  CASE lgcIdx OF
   1: phyIdx := 33;
   2: phyIdx := 34;
   3: phyIdx := 35;
   4: phyIdx := 36;
   5: phyIdx := 37;
   6: phyIdx := 38;
   7: phyIdx := 39;
   8: phyIdx := 40;
   9: phyIdx := 41;
   10: phyIdx := 42;
  END_CASE;
 ELSE
  level := 0;
  phyIdx := 0;
  direct := TargetDirect.undefined;
END_CASE;
END_FUNCTION_BLOCK

(* ---- mdbsLogicToPhy_3.st ---- *)
FUNCTION_BLOCK mdbsLogicToPhy	//modbus华中挡板地址编号对应本地索引编号
VAR_INPUT
section		:INT;	//区域限定 1:skyExt, 2:skyRet, 3:grdExt, 4:grdRet)
lgcIdx		:INT;	//华中对应的地址	10,14{1..10}  17,20{1..11}
END_VAR
VAR_OUTPUT
level		:INT;	//1->地轨	2->天轨
phyIdx		:INT;	//内存物理地址对应数组索引
direct		:TargetDirect;
END_VAR

CASE section OF
1: // skyExtend
 level := 2;
 direct := TargetDirect.extend;
 CASE lgcIdx OF
 1: phyIdx := 1;
 2: phyIdx := 3;
 3: phyIdx := 4;
 4: phyIdx := 5;
 5: phyIdx := 6;
 6: phyIdx := 8;
 7: phyIdx := 9;
 8: phyIdx := 10;
 9: phyIdx := 11;
 10: phyIdx := 12;
 END_CASE;
2: // skyRetract
 level := 2;
 direct := TargetDirect.retract;
 CASE lgcIdx OF
 1: phyIdx := 13;
 2: phyIdx := 14;
 3: phyIdx := 15;
 4: phyIdx := 16;
 5: phyIdx := 17;
 6: phyIdx := 18;
 7: phyIdx := 19;
 8: phyIdx := 20;
 9: phyIdx := 21;
 10: phyIdx := 22;
 END_CASE;
3: // groundExtend
 level := 1;
 direct := TargetDirect.extend;
 CASE lgcIdx OF
 1: phyIdx := 23;
 2: phyIdx := 24;
 3: phyIdx := 25;
 4: phyIdx := 26;
 5: phyIdx := 27;
 6: phyIdx := 28;
 7: phyIdx := 29;
 8: phyIdx := 30;
 9: phyIdx := 31;
 10: phyIdx := 32;
 END_CASE;
4: // groundRetract
 level := 1;
 direct := TargetDirect.retract;
 CASE lgcIdx OF
 1: phyIdx := 33;
 2: phyIdx := 34;
 3: phyIdx := 35;
 4: phyIdx := 36;
 5: phyIdx := 37;
 6: phyIdx := 38;
 7: phyIdx := 39;
 8: phyIdx := 40;
 9: phyIdx := 41;
 10: phyIdx := 42;
 END_CASE;
ELSE
 level := 0;
 phyIdx := 0;
 direct := TargetDirect.undefined;
END_CASE;
END_FUNCTION_BLOCK

(* ---- mdbsNumToIdx_0.st ---- *)
FUNCTION_BLOCK mdbsNumToIdx
VAR_INPUT
	devNo		:WORD;
END_VAR
VAR_OUTPUT
	level		:INT;
	idx			:INT;
END_VAR
VAR
END_VAR

IF devNo > 40000 THEN
	CASE devNo OF
		// 地轨 Level 1
		41010:	level := 1;	idx := 1;
		41020:	level := 1;	idx := 3;
		41030:	level := 1;	idx := 4;
		41040:	level := 1;	idx := 5;
		41050:	level := 1;	idx := 6;
		41060:	level := 1;	idx := 8;
		41070:	level := 1;	idx := 9;
		41080:	level := 1;	idx := 10;
		42010:	level := 1;	idx := 2;
		42020:	level := 1;	idx := 7;

		// 地轨 Level 2
		51010:	level := 2;	idx := 1;
		51020:	level := 2;	idx := 3;
		51030:	level := 2;	idx := 4;
		51040:	level := 2;	idx := 5;
		51050:	level := 2;	idx := 6;
		51060:	level := 2;	idx := 8;
		51070:	level := 2;	idx := 9;
		51080:	level := 2;	idx := 10;
		52010:	level := 2;	idx := 2;
		52020:	level := 2;	idx := 7;

		// 地轨 Level 3
		61010:	level := 3;	idx := 1;
		61020:	level := 3;	idx := 3;
		61030:	level := 3;	idx := 4;
		61040:	level := 3;	idx := 5;
		61050:	level := 3;	idx := 6;
		61060:	level := 3;	idx := 8;
		61070:	level := 3;	idx := 9;
		61080:	level := 3;	idx := 10;
		62010:	level := 3;	idx := 2;
		62020:	level := 3;	idx := 7;

		// Default case
		ELSE
			level := -1;	idx := -1;
	END_CASE;
ELSE
	level := -1;	idx := -1;
END_IF;
END_FUNCTION_BLOCK

(* ---- mdbsNumToIdx_1.st ---- *)
FUNCTION_BLOCK mdbsNumToIdx
VAR_INPUT
	devNo		:WORD;
END_VAR
VAR_OUTPUT
	level		:INT;
	idx			:INT;
END_VAR
VAR
END_VAR

IF devNo > 40000 THEN
  CASE devNo OF
    // 地轨 Level 1
    41010:	level := 1;	idx := 1;
    41020:	level := 1;	idx := 3;
    41030:	level := 1;	idx := 4;
    41040:	level := 1;	idx := 5;
    41050:	level := 1;	idx := 6;
    41060:	level := 1;	idx := 8;
    41070:	level := 1;	idx := 9;
    41080:	level := 1;	idx := 10;
    42010:	level := 1;	idx := 2;
    42020:	level := 1;	idx := 7;

    // 地轨 Level 2
    51010:	level := 2;	idx := 1;
    51020:	level := 2;	idx := 3;
    51030:	level := 2;	idx := 4;
    51040:	level := 2;	idx := 5;
    51050:	level := 2;	idx := 6;
    51060:	level := 2;	idx := 8;
    51070:	level := 2;	idx := 9;
    51080:	level := 2;	idx := 10;
    52010:	level := 2;	idx := 2;
    52020:	level := 2;	idx := 7;

    // 地轨 Level 3
    61010:	level := 3;	idx := 1;
    61020:	level := 3;	idx := 3;
    61030:	level := 3;	idx := 4;
    61040:	level := 3;	idx := 5;
    61050:	level := 3;	idx := 6;
    61060:	level := 3;	idx := 8;
    61070:	level := 3;	idx := 9;
    61080:	level := 3;	idx := 10;
    62010:	level := 3;	idx := 2;
    62020:	level := 3;	idx := 7;

    // Default case
    ELSE
      level := -1;	idx := -1;
  END_CASE;
ELSE
  level := -1;	idx := -1;
END_IF;
END_FUNCTION_BLOCK

(* ---- mdbsNumToIdx_3.st ---- *)
FUNCTION_BLOCK mdbsNumToIdx
VAR_INPUT
	devNo		:WORD;
END_VAR
VAR_OUTPUT
	level		:INT;
	idx			:INT;
END_VAR
(* Removed the empty VAR section as it serves no purpose. This cleanup is not strictly required but is recommended for clarity and adherence to best practices. *)

IF devNo > 40000 THEN
  CASE devNo OF
    // 地轨 Level 1
    41010:	level := 1;	idx := 1;
    41020:	level := 1;	idx := 3;
    41030:	level := 1;	idx := 4;
    41040:	level := 1;	idx := 5;
    41050:	level := 1;	idx := 6;
    41060:	level := 1;	idx := 8;
    41070:	level := 1;	idx := 9;
    41080:	level := 1;	idx := 10;
    42010:	level := 1;	idx := 2;
    42020:	level := 1;	idx := 7;

    // 地轨 Level 2
    51010:	level := 2;	idx := 1;
    51020:	level := 2;	idx := 3;
    51030:	level := 2;	idx := 4;
    51040:	level := 2;	idx := 5;
    51050:	level := 2;	idx := 6;
    51060:	level := 2;	idx := 8;
    51070:	level := 2;	idx := 9;
    51080:	level := 2;	idx := 10;
    52010:	level := 2;	idx := 2;
    52020:	level := 2;	idx := 7;

    // 地轨 Level 3
    61010:	level := 3;	idx := 1;
    61020:	level := 3;	idx := 3;
    61030:	level := 3;	idx := 4;
    61040:	level := 3;	idx := 5;
    61050:	level := 3;	idx := 6;
    61060:	level := 3;	idx := 8;
    61070:	level := 3;	idx := 9;
    61080:	level := 3;	idx := 10;
    62010:	level := 3;	idx := 2;
    62020:	level := 3;	idx := 7;

    // Default case
    ELSE
      level := -1;	idx := -1;
  END_CASE;
ELSE
  level := -1;	idx := -1;
END_IF;
END_FUNCTION_BLOCK

(* ---- mdbsPhyToLogic_0.st ---- *)
FUNCTION_BLOCK mdbsPhyToLogic	//modbus本地索引对应回传华中的状态地址
VAR_INPUT
	section		:INT;	//区域限定(1:grdExt, 2:grdRet, 3:skyExt, 4:skyRet)
	phyIdx		:INT;	//内存物理地址对应数组索引
END_VAR
VAR_OUTPUT
	lgcIdx		:INT;	//华中对应的地址	127 175 223 271...
END_VAR
VAR
END_VAR

CASE section OF
    1: // 区域限定(1:groundExtend)
        CASE phyIdx OF
            1:  lgcIdx := 223;  // grd1e -> 横1 223
            2:  lgcIdx := 231;  // grd2e -> 纵1 231
            3:  lgcIdx := 224;  // grd3e -> 横2 224
            4:  lgcIdx := 225;  // grd4e -> 横3 225
            5:  lgcIdx := 226;  // grd5e -> 横4 226
            6:  lgcIdx := 227;  // grd6e -> 横5 227
            7:  lgcIdx := 232;  // grd7e -> 纵2 232
            8:  lgcIdx := 228;  // grd8e -> 横6 228
            9:  lgcIdx := 229;  // grd9e -> 横7 229
            10: lgcIdx := 230;  // grd10e -> 横8 230
        ELSE
            lgcIdx := -1; // 无效索引
        END_CASE
    2: // 区域限定(2:groundRetract)
        CASE phyIdx OF
            1:  lgcIdx := 271;  // grd1r -> 横1 271
            2:  lgcIdx := 279;  // grd2r -> 纵1 279
            3:  lgcIdx := 272;  // grd3r -> 横2 272
            4:  lgcIdx := 273;  // grd4r -> 横3 273
            5:  lgcIdx := 274;  // grd5r -> 横4 274
            6:  lgcIdx := 275;  // grd6r -> 横5 275
            7:  lgcIdx := 280;  // grd7r -> 纵2 280
            8:  lgcIdx := 276;  // grd8r -> 横6 276
            9:  lgcIdx := 277;  // grd9r -> 横7 277
            10: lgcIdx := 278;  // grd10r -> 横8 278
        ELSE
            lgcIdx := -1; // 无效索引
        END_CASE
    3: // 区域限定(3:skyExtend)
        CASE phyIdx OF
            1:  lgcIdx := 127;  // sky1e -> 横1 127
            2:  lgcIdx := 135;  // sky2e -> 纵1 135
            3:  lgcIdx := 128;  // sky3e -> 横2 128
            4:  lgcIdx := 129;  // sky4e -> 横3 129
            5:  lgcIdx := 130;  // sky5e -> 横4 130
            6:  lgcIdx := 131;  // sky6e -> 横5 131
            7:  lgcIdx := 136;  // sky7e -> 纵2 136
            8:  lgcIdx := 132;  // sky8e -> 横6 132
            9:  lgcIdx := 133;  // sky9e -> 横7 133
            10: lgcIdx := 134;  // sky10e -> 横8 134
        ELSE
            lgcIdx := -1; // 无效索引
        END_CASE
    4: // 区域限定(4:skyRetract)
        CASE phyIdx OF
            1:  lgcIdx := 175;  // sky1r -> 横1 175
            2:  lgcIdx := 183;  // sky2r -> 纵1 183
            3:  lgcIdx := 176;  // sky3r -> 横2 176
            4:  lgcIdx := 177;  // sky4r -> 横3 177
            5:  lgcIdx := 178;  // sky5r -> 横4 178
            6:  lgcIdx := 179;  // sky6r -> 横5 179
            7:  lgcIdx := 184;  // sky7r -> 纵2 184
            8:  lgcIdx
END_FUNCTION_BLOCK

(* ---- mdbsPhyToLogic_1.st ---- *)
FUNCTION_BLOCK mdbsPhyToLogic	//modbus本地索引对应回传华中的状态地址
VAR_INPUT
	section		:INT;	//区域限定(1:grdExt, 2:grdRet, 3:skyExt, 4:skyRet)
	phyIdx		:INT;	//内存物理地址对应数组索引
END_VAR
VAR_OUTPUT
	lgcIdx		:INT;	//华中对应的地址	127 175 223 271...
END_VAR
VAR
END_VAR

CASE section OF
    1: // 区域限定(1:groundExtend)
        CASE phyIdx OF
            1:  lgcIdx := 223;  // grd1e -> 横1 223
            2:  lgcIdx := 231;  // grd2e -> 纵1 231
            3:  lgcIdx := 224;  // grd3e -> 横2 224
            4:  lgcIdx := 225;  // grd4e -> 横3 225
            5:  lgcIdx := 226;  // grd5e -> 横4 226
            6:  lgcIdx := 227;  // grd6e -> 横5 227
            7:  lgcIdx := 232;  // grd7e -> 纵2 232
            8:  lgcIdx := 228;  // grd8e -> 横6 228
            9:  lgcIdx := 229;  // grd9e -> 横7 229
            10: lgcIdx := 230;  // grd10e -> 横8 230
        ELSE
            lgcIdx := -1; // 无效索引
        END_CASE
    2: // 区域限定(2:groundRetract)
        CASE phyIdx OF
            1:  lgcIdx := 271;  // grd1r -> 横1 271
            2:  lgcIdx := 279;  // grd2r -> 纵1 279
            3:  lgcIdx := 272;  // grd3r -> 横2 272
            4:  lgcIdx := 273;  // grd4r -> 横3 273
            5:  lgcIdx := 274;  // grd5r -> 横4 274
            6:  lgcIdx := 275;  // grd6r -> 横5 275
            7:  lgcIdx := 280;  // grd7r -> 纵2 280
            8:  lgcIdx := 276;  // grd8r -> 横6 276
            9:  lgcIdx := 277;  // grd9r -> 横7 277
            10: lgcIdx := 278;  // grd10r -> 横8 278
        ELSE
            lgcIdx := -1; // 无效索引
        END_CASE
    3: // 区域限定(3:skyExtend)
        CASE phyIdx OF
            1:  lgcIdx := 127;  // sky1e -> 横1 127
            2:  lgcIdx := 135;  // sky2e -> 纵1 135
            3:  lgcIdx := 128;  // sky3e -> 横2 128
            4:  lgcIdx := 129;  // sky4e -> 横3 129
            5:  lgcIdx := 130;  // sky5e -> 横4 130
            6:  lgcIdx := 131;  // sky6e -> 横5 131
            7:  lgcIdx := 136;  // sky7e -> 纵2 136
            8:  lgcIdx := 132;  // sky8e -> 横6 132
            9:  lgcIdx := 133;  // sky9e -> 横7 133
            10: lgcIdx := 134;  // sky10e -> 横8 134
        ELSE
            lgcIdx := -1; // 无效索引
        END_CASE
    4: // 区域限定(4:skyRetract)
        CASE phyIdx OF
            1:  lgcIdx := 175;  // sky1r -> 横1 175
            2:  lgcIdx := 183;  // sky2r -> 纵1 183
            3:  lgcIdx := 176;  // sky3r -> 横2 176
            4:  lgcIdx := 177;  // sky4r -> 横3 177
            5:  lgcIdx := 178;  // sky5r -> 横4 178
            6:  lgcIdx := 179;  // sky6r -> 横5 179
            7:  lgcIdx := 184;  // sky7r -> 纵2 184
            8:  lgcIdx
END_FUNCTION_BLOCK

(* ---- mdbsPhyToLogic_2.st ---- *)
FUNCTION_BLOCK mdbsPhyToLogic	//modbus本地索引对应回传华中的状态地址
VAR_INPUT
	section		:INT;	//区域限定(1:grdExt, 2:grdRet, 3:skyExt, 4:skyRet)
	phyIdx		:INT;	//内存物理地址对应数组索引
END_VAR
VAR_OUTPUT
	lgcIdx		:INT;	//华中对应的地址	127 175 223 271...
END_VAR
VAR
END_VAR

CASE section OF
    1: // 区域限定(1:groundExtend)
        CASE phyIdx OF
            1:  lgcIdx := 223;  // grd1e -> 横1 223
            2:  lgcIdx := 231;  // grd2e -> 纵1 231
            3:  lgcIdx := 224;  // grd3e -> 横2 224
            4:  lgcIdx := 225;  // grd4e -> 横3 225
            5:  lgcIdx := 226;  // grd5e -> 横4 226
            6:  lgcIdx := 227;  // grd6e -> 横5 227
            7:  lgcIdx := 232;  // grd7e -> 纵2 232
            8:  lgcIdx := 228;  // grd8e -> 横6 228
            9:  lgcIdx := 229;  // grd9e -> 横7 229
            10: lgcIdx := 230;  // grd10e -> 横8 230
        ELSE
            lgcIdx := -1; // 无效索引
        END_CASE
    2: // 区域限定(2:groundRetract)
        CASE phyIdx OF
            1:  lgcIdx := 271;  // grd1r -> 横1 271
            2:  lgcIdx := 279;  // grd2r -> 纵1 279
            3:  lgcIdx := 272;  // grd3r -> 横2 272
            4:  lgcIdx := 273;  // grd4r -> 横3 273
            5:  lgcIdx := 274;  // grd5r -> 横4 274
            6:  lgcIdx := 275;  // grd6r -> 横5 275
            7:  lgcIdx := 280;  // grd7r -> 纵2 280
            8:  lgcIdx := 276;  // grd8r -> 横6 276
            9:  lgcIdx := 277;  // grd9r -> 横7 277
            10: lgcIdx := 278;  // grd10r -> 横8 278
        ELSE
            lgcIdx := -1; // 无效索引
        END_CASE
    3: // 区域限定(3:skyExtend)
        CASE phyIdx OF
            1:  lgcIdx := 127;  // sky1e -> 横1 127
            2:  lgcIdx := 135;  // sky2e -> 纵1 135
            3:  lgcIdx := 128;  // sky3e -> 横2 128
            4:  lgcIdx := 129;  // sky4e -> 横3 129
            5:  lgcIdx := 130;  // sky5e -> 横4 130
            6:  lgcIdx := 131;  // sky6e -> 横5 131
            7:  lgcIdx := 136;  // sky7e -> 纵2 136
            8:  lgcIdx := 132;  // sky8e -> 横6 132
            9:  lgcIdx := 133;  // sky9e -> 横7 133
            10: lgcIdx := 134;  // sky10e -> 横8 134
        ELSE
            lgcIdx := -1; // 无效索引
        END_CASE
4: // 区域限定(4:skyRetract)
    CASE phyIdx OF
      1:  lgcIdx := 175;  // sky1r -> 横1 175
      2:  lgcIdx := 183;  // sky2r -> 纵1 183
      3:  lgcIdx := 176;  // sky3r -> 横2 176
      4:  lgcIdx := 177;  // sky4r -> 横3 177
      5:  lgcIdx := 178;  // sky5r -> 横4 178
      6:  lgcIdx := 179;  // sky6r -> 横5 179
      7:  lgcIdx := 184;  // sky7r -> 纵2 184
      8:  lgcIdx := 180;  // sky8r -> 横6 180
      9:  lgcIdx := 181;  // sky9r -> 横7 181
      10: lgcIdx := 182;  // sky10r -> 横8 182
    ELSE
      lgcIdx := -1; // 无效索引
    END_CASE
END_CASE
END_FUNCTION_BLOCK

(* ---- mdbsPhyToLogic_3.st ---- *)
FUNCTION_BLOCK mdbsPhyToLogic	//modbus本地索引对应回传华中的状态地址
VAR_INPUT
	section		:INT;	//区域限定(1:grdExt, 2:grdRet, 3:skyExt, 4:skyRet)
	phyIdx		:INT;	//内存物理地址对应数组索引
END_VAR
VAR_OUTPUT
	lgcIdx		:INT;	//华中对应的地址	127 175 223 271...
END_VAR
VAR
END_VAR

CASE section OF
    1: // 区域限定(1:groundExtend)
        CASE phyIdx OF
            1:  lgcIdx := 223;  // grd1e -> 横1 223
            2:  lgcIdx := 231;  // grd2e -> 纵1 231
            3:  lgcIdx := 224;  // grd3e -> 横2 224
            4:  lgcIdx := 225;  // grd4e -> 横3 225
            5:  lgcIdx := 226;  // grd5e -> 横4 226
            6:  lgcIdx := 227;  // grd6e -> 横5 227
            7:  lgcIdx := 232;  // grd7e -> 纵2 232
            8:  lgcIdx := 228;  // grd8e -> 横6 228
            9:  lgcIdx := 229;  // grd9e -> 横7 229
            10: lgcIdx := 230;  // grd10e -> 横8 230
        ELSE
            lgcIdx := -1; // 无效索引
        END_CASE
    2: // 区域限定(2:groundRetract)
        CASE phyIdx OF
            1:  lgcIdx := 271;  // grd1r -> 横1 271
            2:  lgcIdx := 279;  // grd2r -> 纵1 279
            3:  lgcIdx := 272;  // grd3r -> 横2 272
            4:  lgcIdx := 273;  // grd4r -> 横3 273
            5:  lgcIdx := 274;  // grd5r -> 横4 274
            6:  lgcIdx := 275;  // grd6r -> 横5 275
            7:  lgcIdx := 280;  // grd7r -> 纵2 280
            8:  lgcIdx := 276;  // grd8r -> 横6 276
            9:  lgcIdx := 277;  // grd9r -> 横7 277
            10: lgcIdx := 278;  // grd10r -> 横8 278
        ELSE
            lgcIdx := -1; // 无效索引
        END_CASE
3: // 区域限定(3:skyExtend)
    CASE phyIdx OF
      1:  lgcIdx := 127;  // sky1e -> 横1 127
      2:  lgcIdx := 135;  // sky2e -> 纵1 135
      3:  lgcIdx := 128;  // sky3e -> 横2 128
      4:  lgcIdx := 129;  // sky4e -> 横3 129
      5:  lgcIdx := 130;  // sky5e -> 横4 130
      6:  lgcIdx := 131;  // sky6e -> 横5 131
      7:  lgcIdx := 136;  // sky7e -> 纵2 136
      8:  lgcIdx := 132;  // sky8e -> 横6 132
      9:  lgcIdx := 133;  // sky9e -> 横7 133
      10: lgcIdx := 134;  // sky10e -> 横8 134
    ELSE
      lgcIdx := -1; // 无效索引
    END_CASE
  END_CASE
  4: // 区域限定(4:skyRetract)
    CASE phyIdx OF
      1:  lgcIdx := 175;  // sky1r -> 横1 175
      2:  lgcIdx := 183;  // sky2r -> 纵1 183
      3:  lgcIdx := 176;  // sky3r -> 横2 176
      4:  lgcIdx := 177;  // sky4r -> 横3 177
      5:  lgcIdx := 178;  // sky5r -> 横4 178
      6:  lgcIdx := 179;  // sky6r -> 横5 179
      7:  lgcIdx := 184;  // sky7r -> 纵2 184
      8:  lgcIdx := 180;  // sky8r -> 横6 180
      9:  lgcIdx := 181;  // sky9r -> 横7 181
      10: lgcIdx := 182;  // sky10r -> 横8 182
    ELSE
      lgcIdx := -1; // 无效索引
    END_CASE
  END_CASE
END_FUNCTION_BLOCK
